(* Logix 5000 project; controller Lab7_Unit18 vendor 1 type 14 code 106 rev 30.11; software revision 30.00 *)

TASK MainTask (continuous, watchdog 500 ms) : MainProgram

MODULES
   Local : vendor 1 type 14 code 106 (Compact 0, rev 30.11)
      I1 : 1769-IQ16 (Compact 1, rev 1.1, Input RPI 20 ms)
      A3 : vendor 1 type 10 code 33 (Compact 3, rev 1.1, Output RPI 80 ms)
      O2 : vendor 1 type 7 code 86 (Compact 2, rev 2.1, Output RPI 20 ms)
END_MODULES

PROGRAM MainProgram   (* main routine MainRoutine *)
VAR
   Black_Mushroomhead_PB : ALIAS FOR Local:1:I.Data.5;
   Blue_Flush_PB : ALIAS FOR Local:1:I.Data.1;
   Blue_Indicator : ALIAS FOR Local:2:O.Data.3;
   Green_Flush_PB : ALIAS FOR Local:1:I.Data.2;
   Green_Indicator : ALIAS FOR Local:2:O.Data.1;
   Machine_Active : BOOL;
   Motor_Enable : ALIAS FOR Local:2:O.Data.0;
   PowerFlex_Forward : ALIAS FOR Local:2:O.Data.6;
   PowerFlex_Reverse : ALIAS FOR Local:2:O.Data.7;
   Red_Flush_PB : ALIAS FOR Local:1:I.Data.4;
   Red_Indicator : ALIAS FOR Local:2:O.Data.5;
   Red_Mushroomhead_PB : ALIAS FOR Local:1:I.Data.6;
   White_Flush_PB : ALIAS FOR Local:1:I.Data.0;
   White_Indicator : ALIAS FOR Local:2:O.Data.4;
   Yellow_Flush_PB : ALIAS FOR Local:1:I.Data.3;
   Yellow_Indicator : ALIAS FOR Local:2:O.Data.2;
END_VAR

ROUTINE Forward   (* ladder *)
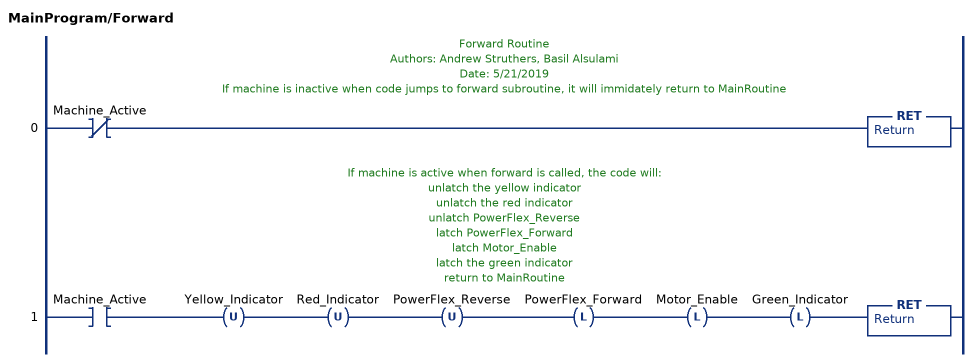
   // Forward Routine
   // Authors: Andrew Struthers, Basil Alsulami
   // Date: 5/21/2019
   // If machine is inactive when code jumps to forward subroutine, it will immidately return to MainRoutine
   0: XIO(Machine_Active)RET();
   // If machine is active when forward is called, the code will:
   // unlatch the yellow indicator
   // unlatch the red indicator
   // unlatch PowerFlex_Reverse
   // latch PowerFlex_Forward
   // latch Motor_Enable
   // latch the green indicator
   // return to MainRoutine
   1: XIC(Machine_Active)OTU(Yellow_Indicator)OTU(Red_Indicator)OTU(PowerFlex_Reverse)OTL(PowerFlex_Forward)OTL(Motor_Enable)OTL(Green_Indicator)RET();
END_ROUTINE

ROUTINE MainRoutine   (* ladder *)
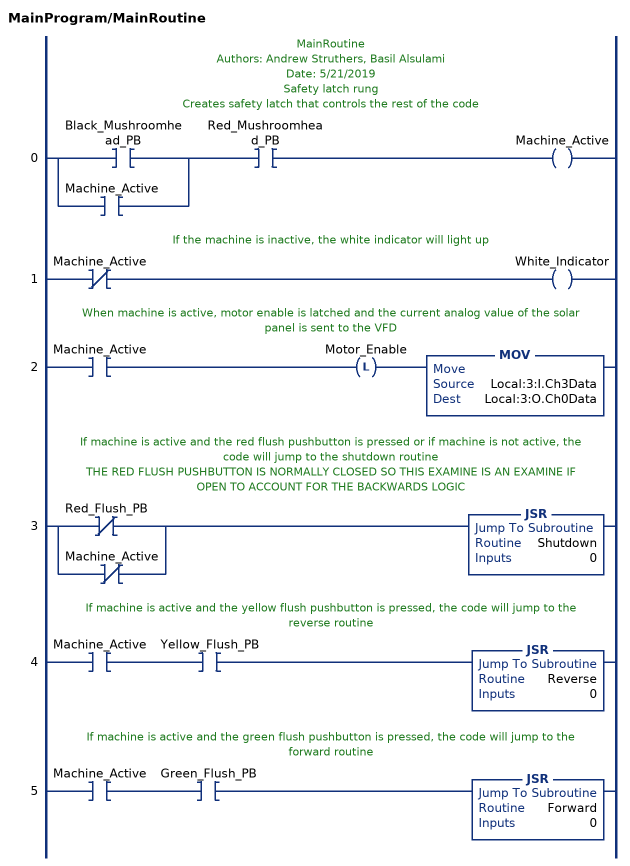
   // MainRoutine
   // Authors: Andrew Struthers, Basil Alsulami
   // Date: 5/21/2019
   // Safety latch rung
   // Creates safety latch that controls the rest of the code
   0: [XIC(Black_Mushroomhead_PB) ,XIC(Machine_Active) ]XIC(Red_Mushroomhead_PB)OTE(Machine_Active);
   // If the machine is inactive, the white indicator will light up
   1: XIO(Machine_Active)OTE(White_Indicator);
   // When machine is active, motor enable is latched and the current analog value of the solar panel is sent to the VFD
   2: XIC(Machine_Active)OTL(Motor_Enable)MOV(Local:3:I.Ch3Data,Local:3:O.Ch0Data);
   // If machine is active and the red flush pushbutton is pressed or if machine is not active, the code will jump to the shutdown routine
   // THE RED FLUSH PUSHBUTTON IS NORMALLY CLOSED SO THIS EXAMINE IS AN EXAMINE IF OPEN TO ACCOUNT FOR THE BACKWARDS LOGIC
   3: [XIO(Red_Flush_PB) ,XIO(Machine_Active) ]JSR(Shutdown,0);
   // If machine is active and the yellow flush pushbutton is pressed, the code will jump to the reverse routine
   4: XIC(Machine_Active)XIC(Yellow_Flush_PB)JSR(Reverse,0);
   // If machine is active and the green flush pushbutton is pressed, the code will jump to the forward routine
   5: XIC(Machine_Active)XIC(Green_Flush_PB)JSR(Forward,0);
END_ROUTINE

ROUTINE Reverse   (* ladder *)
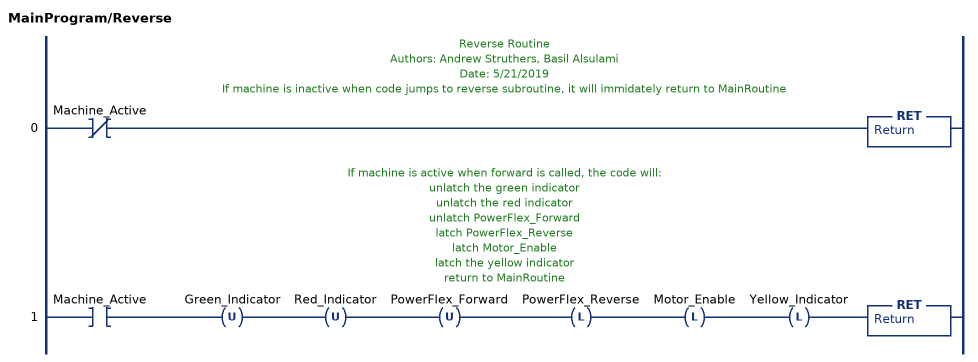
   // Reverse Routine
   // Authors: Andrew Struthers, Basil Alsulami
   // Date: 5/21/2019
   // If machine is inactive when code jumps to reverse subroutine, it will immidately return to MainRoutine
   0: XIO(Machine_Active)RET();
   // If machine is active when forward is called, the code will:
   // unlatch the green indicator
   // unlatch the red indicator
   // unlatch PowerFlex_Forward
   // latch PowerFlex_Reverse
   // latch Motor_Enable
   // latch the yellow indicator
   // return to MainRoutine
   1: XIC(Machine_Active)OTU(Green_Indicator)OTU(Red_Indicator)OTU(PowerFlex_Forward)OTL(PowerFlex_Reverse)OTL(Motor_Enable)OTL(Yellow_Indicator)RET();
END_ROUTINE

ROUTINE Shutdown   (* ladder *)
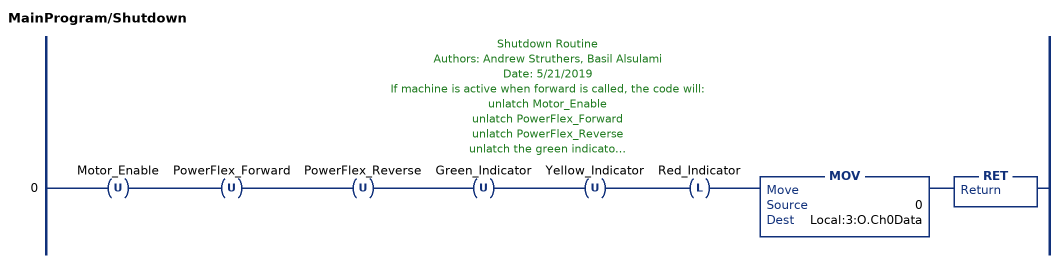
   // Shutdown Routine
   // Authors: Andrew Struthers, Basil Alsulami
   // Date: 5/21/2019
   // If machine is active when forward is called, the code will:
   // unlatch Motor_Enable
   // unlatch PowerFlex_Forward
   // unlatch PowerFlex_Reverse
   // unlatch the green indicator
   // unlatch the yellow indicator
   // latch the red indicator
   // move 0 indo the motor speed bit
   // return to MainRoutine
   0: OTU(Motor_Enable)OTU(PowerFlex_Forward)OTU(PowerFlex_Reverse)OTU(Green_Indicator)OTU(Yellow_Indicator)OTL(Red_Indicator)MOV(0,Local:3:O.Ch0Data)RET();
END_ROUTINE
END_PROGRAM
